// TIA Portal V17 export
// export: Created 2026-04-13T11:12:52.5727938Z, ExportSetting WithDefaults, DisplayName Totally Integrated Automation Portal, DisplayVersion V17 Update 4, DisplayName TIA Portal Openness, DisplayVersion V17 Update 4, DisplayName TIA Portal Version Control Interface, DisplayVersion V17, DisplayName SINAMICS Startdrive Advanced, DisplayVersion V17, DisplayName SINAMICS Startdrive G130, G150, S120, S150, SINAMICS MV, S210, DisplayVersion V17, DisplayName SINAMICS Startdrive G110M, G120, G120C, G120D, G120P, G115D, DisplayVersion V17, DisplayName STEP 7 Professional, DisplayVersion V17 Update 4, DisplayName STEP 7 Safety, DisplayVersion V17, DisplayName WinCC Professional, DisplayVersion V17 Update 4
TagTable "OUTCIPCS2"
  OUTCIPCS2_1设定时间 : Real  (PLC tag OUTCIPCS2.1设定时间, HMI_连接_1, 1 s)
  OUTCIPCS2_2设定时间 : Real  (PLC tag OUTCIPCS2.2设定时间, HMI_连接_1, 1 s)
  OUTCIPCS2_3设定时间 : Real  (PLC tag OUTCIPCS2.3设定时间, HMI_连接_1, 1 s)
  OUTCIPCS2_4设定时间 : Real  (PLC tag OUTCIPCS2.4设定时间, HMI_连接_1, 1 s)
  OUTCIPCS2_5设定时间 : Real  (PLC tag OUTCIPCS2.5设定时间, HMI_连接_1, 1 s)
  OUTCIPCS2_6设定时间 : Real  (PLC tag OUTCIPCS2.6设定时间, HMI_连接_1, 1 s)
  OUTCIPCS2_7设定时间 : Real  (PLC tag OUTCIPCS2.7设定时间, HMI_连接_1, 1 s)
  OUTCIPCS2_8设定时间 : Real  (PLC tag OUTCIPCS2.8设定时间, HMI_连接_1, 1 s)
  OUTCIPCS2_9设定时间 : Real  (PLC tag OUTCIPCS2.9设定时间, HMI_连接_1, 1 s)
  OUTCIPCS2_10设定时间 : Real  (PLC tag OUTCIPCS2.10设定时间, HMI_连接_1, 1 s)
  OUTCIPCS2_11设定时间 : Real  (PLC tag OUTCIPCS2.11设定时间, HMI_连接_1, 1 s)
  OUTCIPCS2_12设定时间 : Real  (PLC tag OUTCIPCS2.12设定时间, HMI_连接_1, 1 s)
  OUTCIPCS2_13设定时间 : Real  (PLC tag OUTCIPCS2.13设定时间, HMI_连接_1, 1 s)
  OUTCIPCS2_14设定时间 : Real  (PLC tag OUTCIPCS2.14设定时间, HMI_连接_1, 1 s)
  OUTCIPCS2_15设定时间 : Real  (PLC tag OUTCIPCS2.15设定时间, HMI_连接_1, 1 s)
  OUTCIPCS2_16设定时间 : Real  (PLC tag OUTCIPCS2.16设定时间, HMI_连接_1, 1 s)
  OUTCIPCS2_1计时 : Real  (PLC tag OUTCIPCS2.1计时, HMI_连接_1, 1 s)
  OUTCIPCS2_2计时 : Real  (PLC tag OUTCIPCS2.2计时, HMI_连接_1, 1 s)
  OUTCIPCS2_3计时 : Real  (PLC tag OUTCIPCS2.3计时, HMI_连接_1, 1 s)
  OUTCIPCS2_4计时 : Real  (PLC tag OUTCIPCS2.4计时, HMI_连接_1, 1 s)
  OUTCIPCS2_5计时 : Real  (PLC tag OUTCIPCS2.5计时, HMI_连接_1, 1 s)
  OUTCIPCS2_6计时 : Real  (PLC tag OUTCIPCS2.6计时, HMI_连接_1, 1 s)
  OUTCIPCS2_7计时 : Real  (PLC tag OUTCIPCS2.7计时, HMI_连接_1, 1 s)
  OUTCIPCS2_8计时 : Real  (PLC tag OUTCIPCS2.8计时, HMI_连接_1, 1 s)
  OUTCIPCS2_9计时 : Real  (PLC tag OUTCIPCS2.9计时, HMI_连接_1, 1 s)
  OUTCIPCS2_10计时 : Real  (PLC tag OUTCIPCS2.10计时, HMI_连接_1, 1 s)
  OUTCIPCS2_11计时 : Real  (PLC tag OUTCIPCS2.11计时, HMI_连接_1, 1 s)
  OUTCIPCS2_12计时 : Real  (PLC tag OUTCIPCS2.12计时, HMI_连接_1, 1 s)
  OUTCIPCS2_13计时 : Real  (PLC tag OUTCIPCS2.13计时, HMI_连接_1, 1 s)
  OUTCIPCS2_14计时 : Real  (PLC tag OUTCIPCS2.14计时, HMI_连接_1, 1 s)
  OUTCIPCS2_15计时 : Real  (PLC tag OUTCIPCS2.15计时, HMI_连接_1, 1 s)
  OUTCIPCS2_16计时 : Real  (PLC tag OUTCIPCS2.16计时, HMI_连接_1, 1 s)
  OUTCIPCS2_1电导率 : Real  (PLC tag OUTCIPCS2.1电导率, HMI_连接_1, 1 s)
  OUTCIPCS2_2电导率 : Real  (PLC tag OUTCIPCS2.2电导率, HMI_连接_1, 1 s)
  OUTCIPCS2_3电导率 : Real  (PLC tag OUTCIPCS2.3电导率, HMI_连接_1, 1 s)
  OUTCIPCS2_4电导率 : Real  (PLC tag OUTCIPCS2.4电导率, HMI_连接_1, 1 s)
  OUTCIPCS2_5电导率 : Real  (PLC tag OUTCIPCS2.5电导率, HMI_连接_1, 1 s)
  OUTCIPCS2_6电导率 : Real  (PLC tag OUTCIPCS2.6电导率, HMI_连接_1, 1 s)
  OUTCIPCS2_7电导率 : Real  (PLC tag OUTCIPCS2.7电导率, HMI_连接_1, 1 s)
  OUTCIPCS2_8电导率 : Real  (PLC tag OUTCIPCS2.8电导率, HMI_连接_1, 1 s)
  OUTCIPCS2_9电导率 : Real  (PLC tag OUTCIPCS2.9电导率, HMI_连接_1, 1 s)
  OUTCIPCS2_10电导率 : Real  (PLC tag OUTCIPCS2.10电导率, HMI_连接_1, 1 s)
  OUTCIPCS2_11电导率 : Real  (PLC tag OUTCIPCS2.11电导率, HMI_连接_1, 1 s)
  OUTCIPCS2_12电导率 : Real  (PLC tag OUTCIPCS2.12电导率, HMI_连接_1, 1 s)
  OUTCIPCS2_13电导率 : Real  (PLC tag OUTCIPCS2.13电导率, HMI_连接_1, 1 s)
  OUTCIPCS2_14电导率 : Real  (PLC tag OUTCIPCS2.14电导率, HMI_连接_1, 1 s)
  OUTCIPCS2_15电导率 : Real  (PLC tag OUTCIPCS2.15电导率, HMI_连接_1, 1 s)
  OUTCIPCS2_16电导率 : Real  (PLC tag OUTCIPCS2.16电导率, HMI_连接_1, 1 s)
  OUTCIPCS2_1清洗状态 : Bool  (PLC tag OUTCIPCS2.1清洗状态, HMI_连接_1, 1 s)
  OUTCIPCS2_2清洗状态 : Bool  (PLC tag OUTCIPCS2.2清洗状态, HMI_连接_1, 1 s)
  OUTCIPCS2_3清洗状态 : Bool  (PLC tag OUTCIPCS2.3清洗状态, HMI_连接_1, 1 s)
  OUTCIPCS2_4清洗状态 : Bool  (PLC tag OUTCIPCS2.4清洗状态, HMI_连接_1, 1 s)
  OUTCIPCS2_5清洗状态 : Bool  (PLC tag OUTCIPCS2.5清洗状态, HMI_连接_1, 1 s)
  OUTCIPCS2_6清洗状态 : Bool  (PLC tag OUTCIPCS2.6清洗状态, HMI_连接_1, 1 s)
  OUTCIPCS2_7清洗状态 : Bool  (PLC tag OUTCIPCS2.7清洗状态, HMI_连接_1, 1 s)
  OUTCIPCS2_8清洗状态 : Bool  (PLC tag OUTCIPCS2.8清洗状态, HMI_连接_1, 1 s)
  OUTCIPCS2_9清洗状态 : Bool  (PLC tag OUTCIPCS2.9清洗状态, HMI_连接_1, 1 s)
  OUTCIPCS2_10清洗状态 : Bool  (PLC tag OUTCIPCS2.10清洗状态, HMI_连接_1, 1 s)
  OUTCIPCS2_11清洗状态 : Bool  (PLC tag OUTCIPCS2.11清洗状态, HMI_连接_1, 1 s)
  OUTCIPCS2_12清洗状态 : Bool  (PLC tag OUTCIPCS2.12清洗状态, HMI_连接_1, 1 s)
  OUTCIPCS2_13清洗状态 : Bool  (PLC tag OUTCIPCS2.13清洗状态, HMI_连接_1, 1 s)
  OUTCIPCS2_14清洗状态 : Bool  (PLC tag OUTCIPCS2.14清洗状态, HMI_连接_1, 1 s)
  OUTCIPCS2_15清洗状态 : Bool  (PLC tag OUTCIPCS2.15清洗状态, HMI_连接_1, 1 s)
  OUTCIPCS2_16清洗状态 : Bool  (PLC tag OUTCIPCS2.16清洗状态, HMI_连接_1, 1 s)
